# EPICS autosave request: ipApp/Db/MKS651C_settings.req
$(P)$(R)DescA
$(P)$(R)DescB
$(P)$(R)DescC
$(P)$(R)DescD
$(P)$(R)DescE

$(P)$(R)wSetpointA
$(P)$(R)wSetpointB
$(P)$(R)wSetpointC
$(P)$(R)wSetpointD
$(P)$(R)wSetpointE

$(P)$(R)wTypeA
$(P)$(R)wTypeB
$(P)$(R)wTypeC
$(P)$(R)wTypeD
$(P)$(R)wTypeE

$(P)$(R)wSpeedA
$(P)$(R)wSpeedB
$(P)$(R)wSpeedC
$(P)$(R)wSpeedD
$(P)$(R)wSpeedE

$(P)$(R)wLeadA
$(P)$(R)wLeadB
$(P)$(R)wLeadC
$(P)$(R)wLeadD
$(P)$(R)wLeadE

$(P)$(R)wGainA
$(P)$(R)wGainB
$(P)$(R)wGainC
$(P)$(R)wGainD
$(P)$(R)wGainE
